// TwinCAT 3 PLC project Name
// ProgramVersion: 3.1.4026.17
// CompilerDefines: VISU_USEPROPERTYINFO
// libraries:
//   CmpBitmapPool, * (System)
//   Tc2_Standard, * (Beckhoff Automation GmbH)
//   Tc2_System, * (Beckhoff Automation GmbH)
//   Tc2_Utilities, * (Beckhoff Automation GmbH)
//   TextListUtils, * (System)
//   VisuDialogs, * (System)
//   VisuSymbols, 4.5.0.0 (System)
// project tree:
//   DUTs/ DUT_AlarmInfo.TcDUT (not stored), DUT_ProductData.TcDUT (not stored), DUT_ModelData.TcDUT
//   / GlobalTextList.TcGTLO, PlcTask.TcTTO (not stored), Visualization Manager.TcVMO (not stored)
//   GVLs/ GVL_HMI.TcGVL, GVL_Retain.TcGVL, GVL_Status.TcGVL
//   POUs/70_Data/ DataShift.TcPOU
//   POUs/80_HMI/ HMI.TcPOU
//   POUs/99_FB/ fbAlarm.TcPOU
//   POUs/ MAIN.TcPOU, Test.TcPOU
//   VISUs/ ImagePool.TcIPO (not stored), TextList.TcTLO (not stored)
//   VISUs/03_SideFrame/ LowerBar.TcVIS (not stored), SideBar.TcVIS (not stored), UpperBar.TcVIS (not stored)
//   VISUs/02_MainFrame/ Main.TcVIS (not stored), Data.TcVIS (not stored), Alarm.TcVIS, Setting.TcVIS (not stored), Manual.TcVIS (not stored), Model.TcVIS, AstModel.TcVIS
//   VISUs/01_Page/ BasePage.TcVIS
// real-time tasks:
//   TASK PlcTask: cycle T#10ms, priority 21, ADS port 351

// ---- DUTs/DUT_ModelData.TcDUT
TYPE DUT_ModelData :
STRUCT
    sName : STRING; // Model name
    iNumber : INT;  // Model identifier
END_STRUCT
END_TYPE

// ---- GVLs/GVL_HMI.TcGVL
//{attribute 'qualified_only'}
VAR_GLOBAL
	
	iSelectProductNo	: UINT; // Select Product No.
	bSaveProductData	: BOOL;
	bDeleteProductData	: BOOL;
	iSelectRecipeNo		: UINT;
	bSaveRecipeData		: BOOL;
	bDeleteRecipeData	: BOOL;
	bRemoveProductData	: BOOL;
	sCurrentTime		: STRING;
	
// Button
	bBtAutoMode			: BOOL;
	bBtStart			: BOOL;
	bBtStop				: BOOL;
	bBtHome				: BOOL;
	bBtDoorLock			: BOOL;
	bBtDoorUnlock		: BOOL;
	bBtAlarmReset		: BOOL;

// Lamp
	bLpBlink			: BOOL;
	bLpHome				: BOOL;
	bLpAlarmReset		: BOOL;
	bLpAutoMode			: BOOL;
	bLpStart			: BOOL;
	
// Index
	iTextIndex			: INT;	// By 'TextList' 0= Manual, 1= Auto
	iMainFrame			: INT; // 0= Main, 1= Manual, 2= Setting, 3= Model, 4= Data, 5= Alarm

// Frame Number

    bMainScreen			: BOOL;
    bManualScreen		: BOOL;
	bSettingScreen		: BOOL;
	bModelScreen		: BOOL;
	bDataScreen			: BOOL;
	bAlarmScreen		: BOOL;
	
// Message Box
	
	sCurrentTitle		: STRING;
	sCurrentMessage		: STRING;
	bCallMessageBox		: BOOL;


// Test Bt
	bTest				: BOOL;
END_VAR

// ---- GVLs/GVL_Retain.TcGVL
//{attribute 'qualified_only'}
  {attribute 'TcPersistent'}
VAR_GLOBAL
	//Product Data
	astProductData 		: ARRAY[0..cMaxStationNo+1] OF DUT_ProductData;
	astModel                : ARRAY[0..9] OF DUT_ModelData; // Model list
	abMoveShift			: ARRAY[0..cMaxStationNo] OF BOOL;
	// Alarm
	astAlarmHistory		: ARRAY[0..cMaxAlarmLogCount-1] OF DUT_AlarmInfo; // 최근 100개 알람 저장
END_VAR

VAR_GLOBAL CONSTANT
	cMaxAlarmLogCount	: INT := 100; 
	cMaxStationNo 		: INT := 30;
END_VAR

// ---- GVLs/GVL_Status.TcGVL
//{attribute 'qualified_only'}
VAR_GLOBAL
	//DataShift
		fbLocalTime 		: FB_LocalSystemTime;
		
	//Status
		bAutoMode				:BOOL;
		bManualMode				:BOOL;
		bHomeMode				:BOOL;
		bAutoBusy				:BOOL;
		bHomeBusy				:BOOL;
		bManualBusy				:BOOL;
		bAlarm					:BOOL;
		bWarning				:BOOL;
		bHomeComplete			:BOOL;
		bSafetyDoorLocked		:BOOL;
		bSafetyDoorUnlocked		:BOOL;
		bAlarmReset				: BOOL;
		
	//Command
		bStopCmd		:BOOL;
		bAutoCmd		:BOOL;
		bHomeCmd		:BOOL;
		bDoorUnlockCmd	:BOOL;
		bDoorLockCmd	:BOOL;
		

END_VAR

// ---- POUs/MAIN.TcPOU
PROGRAM MAIN
VAR

END_VAR

DataShift();
HMI();

IF GVL_HMI.bTest THEN
	Test();	
END_IF

END_PROGRAM

// ---- POUs/70_Data/DataShift.TcPOU
PROGRAM DataShift
VAR
	bTestBitStart		:BOOL;
	bTestBitEnd			:BOOL;	
	i					:INT; //loop index

END_VAR


// Calculate process time
	GVL_Status.fbLocalTime(bEnable := TRUE);	// Current Time
	IF bTestBitStart AND GVL_Status.fbLocalTime.bValid THEN
		astProductData[1].dtStartTime := SYSTEMTIME_TO_DT(GVL_Status.fbLocalTime.systemTime);
	END_IF
	IF bTestBitEnd AND GVL_Status.fbLocalTime.bValid THEN
		astProductData[1].dtEndTime := SYSTEMTIME_TO_DT(GVL_Status.fbLocalTime.systemTime);
	END_IF		
	astProductData[1].tProcessTime	:= astProductData[1].dtEndTime - astProductData[1].dtStartTime;

//Remove Total Product Data
	IF GVL_HMI.bRemoveProductData THEN
		FOR i := 0 TO cMaxStationNo DO
			astProductData[i] := astProductData[cMaxStationNo+1];
		END_FOR;
		GVL_HMI.bRemoveProductData := FALSE;
	END_IF

//Data Shift
	FOR i := 1 TO (cMaxStationNo) DO
		IF i > 0 AND i <= cMaxStationNo THEN  // 범위 체크 추가
			IF abMoveShift[i] = TRUE THEN
				astProductData[i] := astProductData[i-1];
				astProductData[i-1] := astProductData[cMaxStationNo+1];
				abMoveShift[i] := FALSE;
			END_IF
		END_IF
	END_FOR;

END_PROGRAM

// ---- POUs/80_HMI/HMI.TcPOU
PROGRAM HMI
VAR
	tonBlink : ton;
	tonAlarmReset : ton;
	Test: fbAlarm;
	bTest1: BOOL;
	Test1: fbAlarm;
	bTest2: BOOL;
END_VAR

// Current Time
	GVL_HMI.sCurrentTime := SYSTEMTIME_TO_STRING( GVL_Status.fbLocalTime.systemTime);

// Select Auto Mode
	IF GVL_Status.bAutoCmd = FALSE AND GVL_Status.bAutoBusy = FALSE AND GVL_Status.bManualBusy = FALSE AND GVL_Status.bHomeBusy = FALSE  THEN
		//Turn On Auto Mode 
        IF GVL_HMI.bBtAutoMode = TRUE AND GVL_Status.bAutoMode = FALSE AND GVL_Status.bSafetyDoorLocked THEN
			GVL_Status.bAutoMode := TRUE;
			GVL_HMI.bBtAutoMode := FALSE;
		END_IF
		//Turn Off Auto Mode
		IF GVL_HMI.bBtAutoMode = TRUE AND GVL_Status.bAutoMode = TRUE  THEN
			GVL_Status.bAutoMode := FALSE;
			GVL_HMI.bBtAutoMode := FALSE;
		END_IF
	ELSE
		GVL_HMI.bBtAutoMode := FALSE;
	END_IF
		
        IF GVL_Status.bSafetyDoorUnlocked OR (NOT bDoorUnlockCmd AND NOT bDoorLockCmd)  THEN
		GVL_HMI.bBtAutoMode := FALSE;
	END_IF
	
	gvl_hmi.bLpAutoMode := GVL_Status.bAutoMode OR ( GVL_HMI.bLpBlink AND GVL_Status.bHomeComplete AND GVL_Status.bHomeMode);
	
// Select Manual Mode
	IF GVL_Status.bAutoMode = FALSE THEN
		GVL_Status.bManualMode := TRUE;
		GVL_HMI.iTextIndex := 0;
	ELSE
		GVL_Status.bManualMode := FALSE;
		GVL_HMI.iTextIndex := 1;
	END_IF
	
// Auto Running
	IF GVL_HMI.bBtStart = TRUE AND GVL_Status.bAutoMode = TRUE AND GVL_Status.bHomeComplete = TRUE AND GVL_Status.bAutoBusy = FALSE AND GVL_Status.bManualBusy = FALSE AND GVL_Status.bHomeBusy = FALSE THEN
		GVL_Status.bAutoCmd := TRUE;
		GVL_HMI.bBtStart := FALSE;
	ELSIF GVL_HMI.bBtStart = TRUE AND GVL_Status.bAutoMode = FALSE THEN
		GVL_HMI.bBtStart := FALSE;
	END_IF
	
	gvl_hmi.bLpStart := GVL_Status.bAutoCmd OR ( GVL_HMI.bLpBlink AND GVL_Status.bHomeComplete AND GVL_Status.bAutoMode AND ( NOT gvl_status.bAlarm AND NOT gvl_status.bWarning));
	
	
// Stop 
	IF GVL_HMI.bBtStop = TRUE AND GVL_Status.bStopCmd = FALSE THEN
		GVL_Status.bStopCmd	:= TRUE;
		GVL_HMI.bBtStop := FALSE;
	END_IF
	
	IF GVL_Status.bStopCmd = TRUE AND GVL_Status.bAutoBusy = FALSE AND GVL_Status.bManualBusy = FALSE AND GVL_Status.bHomeBusy = FALSE THEN
		GVL_Status.bAutoCmd := FALSE;
		GVL_Status.bHomeCmd := FALSE;
		GVL_Status.bStopCmd := FALSE;
		GVL_HMI.bBtStop := FALSE;
	END_IF
	
// Home 
	GVL_Status.bHomeMode := GVL_Status.bSafetyDoorLocked AND GVL_Status.bManualMode;
	
	IF GVL_HMI.bBtHome = TRUE AND GVL_Status.bHomeMode = TRUE AND GVL_Status.bAutoBusy = FALSE AND GVL_Status.bManualBusy = FALSE AND GVL_Status.bHomeBusy = FALSE AND GVL_Status.bAutoCmd = FALSE THEN
		GVL_Status.bHomeCmd := TRUE;
		GVL_HMI.bBtHome := FALSE;
	ELSIF GVL_HMI.bBtHome = TRUE AND GVL_Status.bHomeMode = FALSE THEN
		GVL_HMI.bBtHome := FALSE;
	END_IF
	
	IF GVL_Status.bHomeCmd = TRUE AND GVL_Status.bHomeComplete = TRUE THEN
		GVL_Status.bHomeCmd := FALSE;
	END_IF
	
	// bHomeComplete Reset
		IF GVL_Status.bSafetyDoorUnlocked THEN
			GVL_Status.bHomeComplete := FALSE;
		END_IF
	
		GVL_HMI.bLpHome := GVL_Status.bHomeComplete OR ( NOT GVL_Status.bHomeComplete AND GVL_Status.bHomeMode AND GVL_HMI.bLpBlink);
	
// Door Unlock
	IF GVL_HMI.bBtDoorUnlock AND GVL_Status.bManualMode AND NOT GVL_Status.bManualBusy THEN
		GVL_Status.bDoorUnlockCmd := TRUE;
		GVL_Status.bDoorLockCmd := FALSE;
		GVL_HMI.bBtDoorUnlock := FALSE;
	ELSE
		GVL_HMI.bBtDoorUnlock := FALSE;
	END_IF
	
// Door Lock
	IF GVL_HMI.bBtDoorLock AND GVL_Status.bManualMode AND NOT GVL_Status.bManualBusy THEN
		GVL_Status.bDoorLockCmd := TRUE;
		GVL_Status.bDoorUnlockCmd := FALSE;
		GVL_HMI.bBtDoorLock := FALSE;
	ELSE
		GVL_HMI.bBtDoorLock := FALSE;
	END_IF
	
// Alarm Reset
	IF gvl_hmi.bBtAlarmReset THEN
		GVL_Status.bAlarmReset := TRUE;
		gvl_hmi.bBtAlarmReset := FALSE;
	END_IF
	
	tonAlarmReset(in := GVL_Status.bAlarmReset, pt := T#0.5S);
	
	IF tonAlarmReset.Q THEN
		GVL_Status.bAlarmReset := FALSE;
	END_IF
	
	gvl_hmi.bLpAlarmReset := GVL_Status.bAlarmReset OR (GVL_HMI.bLpBlink AND (gvl_status.bAlarm OR gvl_status.bWarning));
		
// blink
 	tonBlink(in := NOT tonBlink.q , PT := T#500MS);
	
	IF tonBlink.Q THEN
		GVL_HMI.bLpBlink := NOT GVL_HMI.bLpBlink;
	END_IF
	
// Current Screen
	gvl_hmi.bMainScreen := gvl_hmi.iMainFrame = 0;
	gvl_hmi.bManualScreen := gvl_hmi.iMainFrame = 1;
	gvl_hmi.bSettingScreen := gvl_hmi.iMainFrame = 2;
	gvl_hmi.bModelScreen := gvl_hmi.iMainFrame = 3;
	gvl_hmi.bDataScreen := gvl_hmi.iMainFrame = 4;
	gvl_hmi.bAlarmScreen := gvl_hmi.iMainFrame = 5;

END_PROGRAM

// ---- POUs/Test.TcPOU
PROGRAM Test
VAR

	fbTestAlarm1: fbalarm;

	bTes1: BOOL;
	bTest11: BOOL;
	bTestError1: BOOL;
	bTestWarning1: BOOL;
END_VAR

// Door		
	GVL_Status.bSafetyDoorLocked := GVL_Status.bDoorLockCmd;
	GVL_Status.bSafetyDoorUnlocked := GVL_Status.bDoorUnlockCmd;
	
// home
	IF GVL_Status.bHomeCmd THEN
		GVL_Status.bHomeComplete := TRUE;
	END_IF



// Alarm
	fbTestAlarm1(
	bSelectWarning:= bTes1, 
	tDelayTime:= T#1S, 
	bCommand:= TRUE, 
	bAlarmCondition:= bTest11, 
	iAlarmCode:= 1, 
	iPriority:= 1, 
	sAlarmMessage:= 'hello', 
	sLocation:= 'office', 
	bError=> bTestError1, 
	bWarning=> bTestWarning1);

END_PROGRAM

// ---- POUs/99_FB/fbAlarm.TcPOU
FUNCTION_BLOCK fbAlarm	// 
VAR_INPUT
	bSelectWarning	: BOOL;
	tDelayTime	: TIME;
	bCommand	: BOOL;
	bAlarmCondition	: BOOL;
	iAlarmCode	: INT;
	iPriority	: INT;
	sAlarmMessage	: STRING;
	sLocation	: STRING;
END_VAR
VAR_OUTPUT
	bError	: BOOL;
	bWarning	: BOOL;
END_VAR
VAR
	bAlarm	: BOOL;
	triAlarm	: R_Trig;
	triWarning	: R_Trig;
	triError	: R_Trig;
	i: INT;
	stAlarmInfo	: Dut_AlarmInfo;
	tonDelayTimer	: ton;
END_VAR


// Alarm Input
	balarm	:= bCommand AND bAlarmCondition;
	tonDelayTimer(in := balarm, pt :=tDelayTime);

// Alarm History
	triAlarm(clk := tonDelayTimer.Q);
	IF triAlarm.Q THEN
		FOR i := cMaxAlarmLogCount TO 1 BY -1 DO
			astAlarmHistory[i]	:= astAlarmHistory[i-1];
		END_FOR
		stalarminfo.iAlarmCode	:= iAlarmCode;
		stalarminfo.iPriority	:= iPriority;
		stalarminfo.sAlarmMessage	:= sAlarmMessage;
		stalarminfo.sLocation	:= sLocation;
		stalarminfo.tTimeStamp	:= SYSTEMTIME_TO_DT(GVL_Status.fbLocalTime.systemTime);
		astAlarmHistory[0] := stAlarmInfo;
	END_IF

// Alarm Output
	IF tonDelayTimer.Q THEN
		bError := NOT bSelectWarning;
		gvl_status.bAlarm := NOT bSelectWarning;
		bWarning := bSelectWarning;
		gvl_status.bWarning := bSelectWarning;
	END_IF
	
// Alarm Reset
	IF bAlarmReset THEN
		bError := FALSE;
		bWarning := FALSE;
		gvl_status.bAlarm := FALSE;
		gvl_status.bWarning := FALSE;
	END_IF
	
// Call Message Box
	triWarning(clk := gvl_status.bWarning);
	IF triWarning.Q THEN
		sCurrentTitle	:= astAlarmHistory[0].sLocation;
		sCurrentMessage	:= astAlarmHistory[0].sAlarmMessage;
		bCallMessageBox := gvl_status.bWarning;
	END_IF
	
// Change Main Frame to Alarm
	triError(clk := gvl_status.bAlarm);
	IF triError.Q THEN
		iMainFrame := 5;
	END_IF

END_FUNCTION_BLOCK

// ---- GlobalTextList.TcGTLO
TEXTLIST GlobalTextList
  422 = '%.19s' | Korea: '%.19s' | English: '%.19s'
  410 = 'a'
  851 = 'Active'
  609 = 'Alarm'
  662 = 'Alarm Code'
  947 = 'Alarm Page'
  35 = 'Alarm Reset'
  411 = 'AlarmCode'
  22 = 'AlarmMessage'
  147 = 'AlarmReset' | Korea: '초기화'
  23 = 'Alarm_Log'
  557 = 'Arkplus' | Korea: '화면인터페이스' | English: 'Standard_HMI'
  491 = 'Auto Mode'
  808 = 'AutoMode'
  787 = 'b'
  699 = 'Code'
  709 = 'Conveyor'
  122 = 'Data'
  161 = 'Data Page'
  226 = 'Door'
  850 = 'Door Close'
  103 = 'Door Open'
  567 = 'DoorClose'
  271 = 'English' | Korea: '영어' | English: 'English'
  697 = 'fdsafdafsda'
  217 = 'GroupBox'
  279 = 'Home'
  332 = 'Korea' | Korea: '한국어' | English: 'Korea'
  0 = 'Location'
  956 = 'Main'
  707 = 'Main Page'
  301 = 'Manual'
  775 = 'Manual Page'
  83 = 'ManualMode'
  186 = 'Message'
  376 = 'Model'
  313 = 'Model Page'
  536 = 'Parameter'
  403 = 'Priority'
  529 = 'Robot'
  204 = 'SafetyBypass'
  331 = 'Sample'
  239 = 'Setting'
  394 = 'Setting Page'
  849 = 'Standard_HMI' | Korea: '화면인터페이스'
  261 = 'Start'
  606 = 'Stop'
  904 = 'Test'
  272 = 'Time Stamp'
  199 = 'TimeStamp'
  396 = 'TurnTable'
  171 = 'yyyy‑MM‑dd\xa0HH:mm:ss'
END_TEXTLIST

// ---- VISUs/02_MainFrame/Alarm.TcVIS
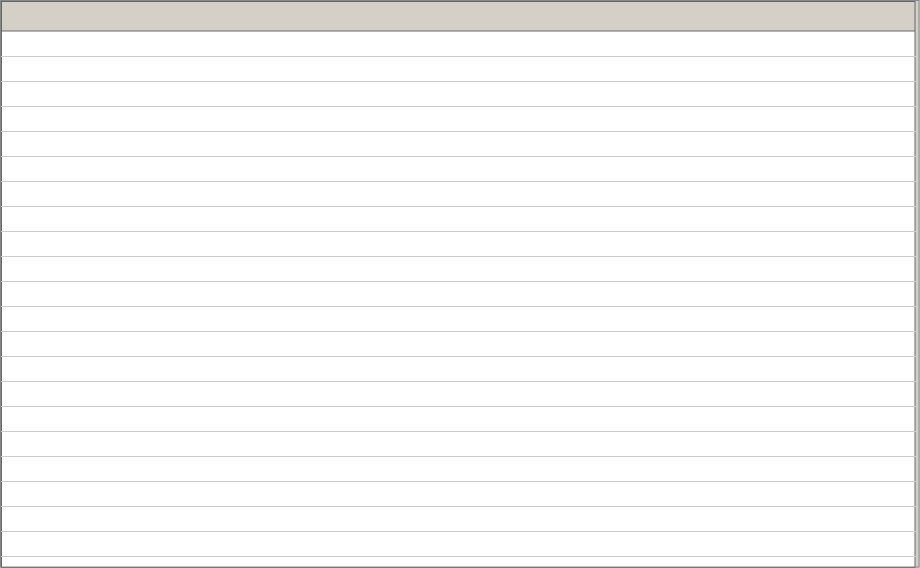
VISUALIZATION Alarm  // 920x568
    Table (1,1 914x567), data array: GVL_Retain.astAlarmHistory
        p3854506369: GVL_Retain.astAlarmHistory[INDEX].bActive
        p1892666644: GVL_Retain.astAlarmHistory[INDEX].iAlarmCode
        p338671338: GVL_Retain.astAlarmHistory[INDEX].sAlarmMessage
        p2170511999: GVL_Retain.astAlarmHistory[INDEX].tTimeStamp
        p3723444502: GVL_Retain.astAlarmHistory[INDEX].sLocation
        p1218418051: GVL_Retain.astAlarmHistory[INDEX].iPriority
        p4092479075: Time Stamp
        p1014161805: 99 - 0 + INT#1
        p1128707560: cMaxAlarmLogCount
END_VISUALIZATION

// ---- VISUs/02_MainFrame/Model.TcVIS
VISUALIZATION Model  // 920x568
END_VISUALIZATION

// ---- VISUs/02_MainFrame/AstModel.TcVIS
VISUALIZATION AstModel  // 2x2
END_VISUALIZATION

// ---- VISUs/01_Page/BasePage.TcVIS
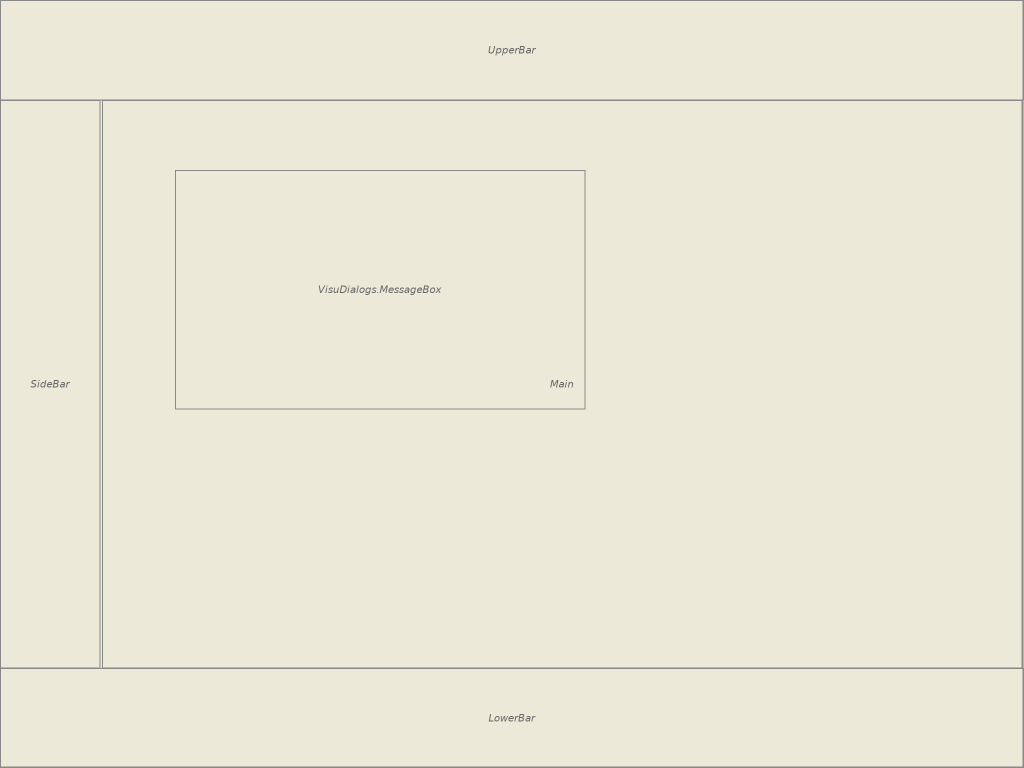
VISUALIZATION BasePage  // 1024x768
    Frame (0,0 1024x100)
        shows UpperBar()
    Frame (0,668 1024x100)
        shows LowerBar()
    Frame (0,100 100x568)
        shows SideBar()
    Frame (102,100 920x568), frame switch variable: GVL_HMI.iMainFrame
        shows Main()
        shows Manual()
        shows Setting()
        shows Model()
        shows Data()
        shows Alarm()
    Frame (175,170 410x239), invisible if: not bCallMessageBox
        shows VisuDialogs.MessageBox(eType := VisuDialogs.MessageBoxDialog_Types.OK_CANCEL, sTitle := sCurrentTitle, sMessageTxt := sCurrentMessage)
        OnMouseClick: execute { bCallMessageBox := false; }
END_VISUALIZATION
